(* IEC 61131-3 sources: structured-text-examples/, 5 files *)

(* ---- backup-generator.st ---- *)
PROGRAM backup_generator
VAR
    X1_0: BOOL; //boilers thermal overload input
    X1_1: BOOL; //water temperature thermal overload input
    X1_2: BOOL; //smog levels exceeded
    Y1_0: BOOL; //main generator
    Y1_1: BOOL; //standby generator

    T_10s: TON; //10 second timer
    rtime: TIME; //5 second timer
    T_5s: TON;
    ztime: TIME;
END_VAR

Y1_0 := X1_0 AND T_10s.Q AND T-5s.Q;
T_10s.IN := X1_1
T_5s.IN := X1_2
Y1_1 := Y1_0

END_PROGRAM

(* ---- blinky_test.st ---- *)
PROGRAM blinky_test
  VAR
    led : BOOL;
    on_timer : TON;
    off_timer : TOF;
  END_VAR

  on_timer.IN := NOT led;
  off_timer.IN := on_timer.Q;
  (* off_timer.PT := T#500ms;
  on_timer.PT := T#500ms;*)
  led := off_timer.Q;
END_PROGRAM

CONFIGURATION Config0

  RESOURCE Res0 ON PLC
    TASK task0(INTERVAL := T#20ms,PRIORITY := 0);
    PROGRAM instance0 WITH task0 : blinky_test;
  END_RESOURCE
END_CONFIGURATION

(* ---- conveyor-belt.st ---- *)
PROGRAM conveyor_belt
VAR
    //inputs
    start_button AT %I0.0: BOOL;
    left_sensor AT %I69.3: BOOL;
    right_sensor AT %I69.4: BOOL;

    //outputs
    stop_button AT %I0.1: BOOL;
    move_left AT %Q65.1: BOOL;
    move_right AT %Q65.0: BOOL;
    should_move_conveyor AT %M0.7: BOOL;
    should_reset AT %M1.0: BOOL;
    increment5 AT %Q0.4: BOOL;
    count AT %QW0: INT;

    //blocks
    counter5 AT %DB6: CTUD;

END_VAR;

should_move_conveyor := start_button OR (should_move_conveyor AND NOT should_reset);
move_left := should_move_conveyor AND (right_sensor OR (move_left AND NOT left_sensor));
move_right := should_move_conveyor AND NOT move_left;
should_reset := increment5 OR stop_button;
update_counter();

FUNCTION update_counter
    counter5.CU := should_move_conveyor AND right_sensor;
    counter5.CD := FALSE;
    counter5.R := should_reset;
    counter5.PV := 5;
    counter5.LD := FALSE;
    increment5 = counter5.QU;
    count := counter5.CV;

END_FUNCTION

END_PROGRAM

(* ---- pwm_servo_attempt.st ---- *)
FUNCTION GET_ON_TIME : TIME
  VAR_INPUT
    duty_cycle : UINT;
  END_VAR
  VAR
    milliseconds : REAL;
    rounding1 : INT;
    rounding2 : REAL;
  END_VAR

  milliseconds := 2.0 / 100.0 * UINT_TO_REAL(duty_cycle);

  (* get all individual unit values *)
  rounding1 := REAL_TO_INT(milliseconds * 100.0);
  rounding2 := INT_TO_REAL(rounding1) / 100000.0;

  (* create string of a real number 2 decimal places *)
  GET_ON_TIME := REAL_TO_TIME(rounding2);
END_FUNCTION

FUNCTION GET_OFF_TIME : TIME
  VAR_INPUT
    duty_cycle : UINT;
  END_VAR
  VAR
    milliseconds : REAL;
    rounding1 : INT;
    rounding2 : REAL;
  END_VAR

  milliseconds := 2.0 - (2.0 / 100.0 * UINT_TO_REAL(duty_cycle));

  (* get all individual unit values *)
  rounding1 := REAL_TO_INT(milliseconds * 100.0);
  rounding2 := INT_TO_REAL(rounding1) / 100000.0;

  (* create string of a real number 2 decimal places *)
  GET_OFF_TIME := REAL_TO_TIME(rounding2);
END_FUNCTION

PROGRAM motor_driver
  VAR
    led AT %QX0.3 : BOOL := true;
  END_VAR
  VAR
    led_on_timer : TON;
    led_off_timer : TOF;
    output_on_timer : TON;
    output_off_timer : TOF;
    input_angle : INT := 90;
    real_angle : REAL := 90.0;
    duty_cycle : UINT := 50;
    on_PT : TIME := T#2ms;
    off_PT : TIME := T#2ms;
  END_VAR
  VAR
    output_pin AT %QW1 : UINT := 65535;
  END_VAR

  (* Blink the builtin LED *)
  led_on_timer(IN := NOT(led_off_timer.Q), PT := T#50ms);
  led_off_timer(IN := led_on_timer.Q, PT := T#50ms);
  led := led_off_timer.Q;

  (* validate the servo angle *)
  IF(input_angle < 0) THEN
    input_angle := 0;

  ELSIF(input_angle > 180) THEN
    input_angle := 180;

  END_IF;

  (* control the servo *)
  real_angle := INT_TO_REAL(input_angle);
  duty_cycle := REAL_TO_UINT(100.0 / 180.0 * real_angle);

  on_PT := GET_ON_TIME(duty_cycle);
  off_PT := GET_OFF_TIME(duty_cycle);

  output_on_timer(IN := NOT(output_off_timer.Q), PT := on_PT);
  output_off_timer(IN := output_on_timer.Q, PT := off_PT);

  IF output_on_timer.Q THEN
    output_pin := 65535;

  ELSE
    output_pin := 0;

  END_IF;
END_PROGRAM

CONFIGURATION Config0

  RESOURCE Res0 ON PLC
    TASK task0(INTERVAL := T#1ms,PRIORITY := 0);
    PROGRAM instance0 WITH task0 : motor_driver;
  END_RESOURCE
END_CONFIGURATION

(* ---- trafficlight-t-intersection.st ---- *)
PROGRAM trafficlight_t_intersection
VAR
    redlight_mainroad AT %Q550.0: BOOL; //red light, main road
    orangelight_mainroad AT %Q550.1: BOOL; //orange light, main road
    greenlight_mainroad AT %Q550.2: BOOL; //green light, main road

    redlight_sidestreet AT %Q550.3: BOOL; //red light, side road
    orangelight_sidestreet AT %Q550.4: BOOL; //orange light, side road
    greenlight_sidestreet AT %Q550.5: BOOL; //green light, side road

    redlight_pedestrian AT %Q550.6: BOOL; //red light pedestrian
    greenlight_pedestrian AT %Q550.7: BOOL; //green light pedestrian

    S1_S2 AT %I500.2: BOOL; //pedestrian button
    S3 AT %I500.5: BOOL; //car sensor induction loop

    SYSTEM_ON AT %I500.0: BOOL; //on switch

    power_state: BOOL
    system_state: INT;
    button_was_pressed: BOOL;
    inducer_was_triggered: BOOL;

    red_timer: TON;
    red_trigger: BOOL;
    yellow_timer: TON;
    yellow_trigger: BOOL;
    green_timer: TON;
    green_trigger: BOOL;

    delay1: TIME := T#3s;
    delay2: TIME := T#10s;
END_VAR

IF SYSTEM_ON THEN
    power_state := TRUE;

ELSE THEN
    power_state := FALSE;
END_IF;

if power_state THEN
    CASE system_state OF
        0: mainroad()
        1: button_pressed()
        2: car_detected()
        3: pedestrians_walk()
        4: sidestreet()
        5: sidestreet_orange()
    END_CASE;

FUNCTION mainroad
    redlight_mainroad := FALSE;
    orangelight_mainroad := FALSE;
    greenlight_mainroad := TRUE;

    redlight_sidestreet := TRUE;
    orangelight_sidestreet := FALSE;
    greenlight_sidestreet := FALSE;

    redlight_pedestrian := TRUE;
    greenlight_pedestrian := FALSE;

    IF S1_S2 = TRUE THEN
        red_timer(IN := red_trigger, PT := delay1);
        red_trigger := TRUE;
        button_was_pressed := TRUE:

    ELSE IF S3 = TRUE THEN
        inducer_was_triggered := TRUE;

    ELSE IF red_timer.Q = TRUE THEN
        red_trigger := FALSE;

        IF button_was_pressed = TRUE THEN
            system_state := 1;
            button_was_pressed := FALSE;

        ELSE IF inducer_was_triggered = TRUE
            system_state := 2;
            inducer_was_triggered := FALSE;

        END_IF;
    END_IF;
END_FUNCTION

FUNCTION mainroad_orange
    VAR_INPUT
        next_state: INT;
    END_VAR;

    greenlight_mainroad := FALSE;
    orangelight_mainroad := TRUE;
    redlight_mainroad := FALSE;

    yellow_timer(IN := yellow_trigger, PT := delay1);
    yellow_trigger := TRUE;

    IF yellow_timer.Q = TRUE THEN
        yellow_trigger := FALSE;
        system_state := next_state;
    END_IF;

END_FUNCTION

FUNCTION button_pressed
    mainroad_orange(3);
END_FUNCTION

FUNCTION car_detected
    mainroad_orange(4);
END_FUNCTION

FUNCTION pedestrians_walk
    greenlight_sidestreet := FALSE;
    orangelight_sidestreet := FALSE;
    redlight_sidestreet := TRUE;

    redlight_pedestrian := FALSE;
    greenlight_pedestrian := TRUE;

    green_timer(IN := green_trigger, PT := delay2);
    green_trigger := TRUE;

    IF green_timer.Q = TRUE THEN
        green_trigger := FALSE;
        system_state := 0;
    END_IF;
END_FUNCTION

FUNCTION sidestreet
    greenlight_mainroad := FALSE;
    orangelight_mainroad := FALSE;
    redlight_mainroad := TRUE;

    greenlight_sidestreet := TRUE;
    orangelight_sidestreet := FALSE;
    redlight_sidestreet := FALSE;

    green_timer(IN := green_trigger, PT := delay2);
    green_trigger := TRUE;

    IF green_timer.Q = TRUE THEN
        green_trigger := FALSE;
        system_state := 5;
    END_IF;
END_FUNCTION

FUNCTION sidestreet_orange
    greenlight_sidestreet := FALSE;
    orangelight_sidestreet := TRUE;
    redlight_sidestreet := FALSE;

    yellow_timer(IN := yellow_trigger, PT := delay1);
    yellow_trigger := TRUE;

    IF yellow_timer.Q = TRUE THEN
        yellow_trigger := FALSE;
        system_state := 0;
    END_IF;
END_FUNCTION

END_PROGRAM
